// TIA Portal V16 export
// export: Created 2021-11-12T13:33:09.7450518Z, ExportSetting WithDefaults, DisplayName Totally Integrated Automation Portal, DisplayVersion V16 Update 3, DisplayName TIA Portal Version Control Interface, DisplayVersion V16 Update 2, DisplayName TIA Portal Openness, DisplayVersion V16 Update 3, DisplayName SINAMICS Startdrive Advanced, DisplayVersion V16 Update 5, DisplayName SINAMICS Startdrive G130, G150, S120, S150, SINAMICS MV, S210, DisplayVersion V16 Update 5, DisplayName SINAMICS Startdrive G110M, G120, G120C, G120D, G120P, G115D, DisplayVersion V16 Update 5, DisplayName STEP 7 Professional, DisplayVersion V16 Update 3, DisplayName STEP 7 Safety, DisplayVersion V16, DisplayName WinCC UA Professional, DisplayVersion V16 Update 3
DATA_BLOCK "IDB_Station440"   // DB218
{ DB_Accessible_From_OPC_UA := 'FALSE' }
VERSION : 0.1
// stored: AutoNumber true, DBAccessibleFromOPCUA false, InstanceOfName Station440, InstanceOfType FB
"Station440"
   // VAR
   //    SF_GL01_MA01 : "STD_Drive1";
   //    SF_UC21_TA1 { S7_SetPoint := 'True'} : "STD_Siemens_G120_CU240E_2_PN";
   //    SF_Alarm1 { S7_SetPoint := 'True'} : "STD_DI_Mon";
   //    SF_Alarm2 { S7_SetPoint := 'True'} : "STD_DI_Mon";
   //    SF_OnOff { S7_SetPoint := 'True'} : "STD_OnOff";
   //    SF_TOF_BSN4 { S7_SetPoint := 'True'} : TOF_TIME;
   //    SB1_PowerOk { S7_SetPoint := 'True'} : Bool;
   // END_VAR
BEGIN
END_DATA_BLOCK
